(* CoDeSys 2.3.9.28 project: moje1.pro *)
(* Libraries: \\psf\Home\Documents\WAGO\libs\library\PowerMeasurement_01.lib 1.1.09 09:28:50, SysLibTime.lib 2.12.10 13:48:32, Building_common.lib 2.12.10 13:48:40, mod_com.lib 2.12.10 13:48:32, Util.lib 18.5.10 14:14:28, Standard.lib 2.12.10 13:48:34, SYSLIBCALLBACK.LIB 2.12.10 13:48:32, \\psf\Home\Documents\WAGO\libs\Libraries_BA\DALI_02.lib 4.3.11 14:50:14 *)

(* PLC configuration (modules and I/O channels)
TL01 AT %IX17.0 [BOOLOnX_I] Vypinac_sklad_sklad
TL02 AT %IX17.1 [BOOLOnX_I] Vypinac_sklad_prodejna
TL03 AT %IX17.2 [BOOLOnX_I] Vypinac_sklad_z_venku
TL04 AT %IX17.3 [BOOLOnX_I] Vypinac_sklad_vrata_predni
TL05 AT %IX17.4 [BOOLOnX_I] Vypinac_sklad_vrata_zadni
TL06 AT %IX17.5 [BOOLOnX_I] Vypinac_prodejna_kolotoc_sude
TL07 AT %IX17.6 [BOOLOnX_I] Vypinac_prodejna_kolotoc_liche
TL08 AT %IX17.7 [BOOLOnX_I] Vypinac_prodejna_vypinac
TL09 AT %IX17.8 [BOOLOnX_I] Prodejna_Dali
TL10 AT %IX17.9 [BOOLOnX_I] Prodejna_faugule_OUT13
TL11 AT %IX17.10 [BOOLOnX_I] Ch_3 Digital input
TL12 AT %IX17.11 [BOOLOnX_I] Ch_4 Digital input
TL13 AT %IX17.12 [BOOLOnX_I] Ch_5 Digital input
AT %IX17.13 [BOOLOnX_I] Ch_6 Digital input
AT %IX17.14 [BOOLOnX_I] Ch_7 Digital input
AT %IX17.15 [BOOLOnX_I] Ch_8 Digital input
0750-0430 8 DI 24 V DC 3.0ms [Type_1_8_Channels] node 2, in %IB2 out %QB2 {INTTypePAAssignment = PLC; INTTypeModule = plugged}
  AT %IX18.0 [BOOLOnX_I] Ch_1 Digital input
  AT %IX18.1 [BOOLOnX_I] Ch_2 Digital input
  AT %IX18.2 [BOOLOnX_I] Ch_3 Digital input
  AT %IX18.3 [BOOLOnX_I] Ch_4 Digital input
  AT %IX18.4 [BOOLOnX_I] Ch_5 Digital input
  AT %IX18.5 [BOOLOnX_I] Ch_6 Digital input
  AT %IX18.6 [BOOLOnX_I] Ch_7 Digital input
  AT %IX18.7 [BOOLOnX_I] Ch_8 Digital input
0750-0530 8 DO 24 V DC 0.5A [Type_10_8_Channels] node 3, in %IB3 out %QB3 {INTTypePAAssignment = PLC; INTTypeModule = plugged}
  KA01 AT %QX9.0 [BOOLOnX_Q] Nevim
  KA02 AT %QX9.1 [BOOLOnX_Q] kolotoc2
  KA03 AT %QX9.2 [BOOLOnX_Q] kolotoc3
  KA04 AT %QX9.3 [BOOLOnX_Q] kolotoc4
  KA05 AT %QX9.4 [BOOLOnX_Q] kolotoc5
  KA06 AT %QX9.5 [BOOLOnX_Q] kolotoc6
  KA07 AT %QX9.6 [BOOLOnX_Q] kolotoc7
  KA08 AT %QX9.7 [BOOLOnX_Q] kolotoc8
0750-0530 8 DO 24 V DC 0.5A [Type_10_8_Channels] node 4, in %IB4 out %QB4 {INTTypePAAssignment = PLC; INTTypeModule = plugged}
  KA09 AT %QX9.8 [BOOLOnX_Q] kolotoc9
  KA10 AT %QX9.9 [BOOLOnX_Q] kolotoc10
  KA11 AT %QX9.10 [BOOLOnX_Q] kolotoc11
  KA12 AT %QX9.11 [BOOLOnX_Q] kolotoc12
  KA13 AT %QX9.12 [BOOLOnX_Q] svetlo_vchod_do_prodejny
  KA14 AT %QX9.13 [BOOLOnX_Q] reklama
  KA15 AT %QX9.14 [BOOLOnX_Q] svetlo_vrata_predni
  KA16 AT %QX9.15 [BOOLOnX_Q] svetlo_vrata_zadni
0750-0530 8 DO 24 V DC 0.5A [Type_10_8_Channels] node 5, in %IB5 out %QB5 {INTTypePAAssignment = PLC; INTTypeModule = plugged}
  KA17 AT %QX10.0 [BOOLOnX_Q] Ch_1 Digital output
  AT %QX10.1 [BOOLOnX_Q] Ch_2 Digital output
  AT %QX10.2 [BOOLOnX_Q] Ch_3 Digital output
  KA20 AT %QX10.3 [BOOLOnX_Q] Ch_4 Digital output
  AT %QX10.4 [BOOLOnX_Q] Ch_5 Digital output
  AT %QX10.5 [BOOLOnX_Q] Ch_6 Digital output
  AT %QX10.6 [BOOLOnX_Q] Ch_7 Digital output
  AT %QX10.7 [BOOLOnX_Q] Ch_8 Digital output
0750-0530 8 DO 24 V DC 0.5A [Type_10_8_Channels] node 6, in %IB6 out %QB6 {INTTypePAAssignment = PLC; INTTypeModule = plugged}
  AT %QX10.8 [BOOLOnX_Q] Ch_1 Digital output
  AT %QX10.9 [BOOLOnX_Q] Ch_2 Digital output
  AT %QX10.10 [BOOLOnX_Q] Ch_3 Digital output
  AT %QX10.11 [BOOLOnX_Q] Ch_4 Digital output
  AT %QX10.12 [BOOLOnX_Q] Ch_5 Digital output
  AT %QX10.13 [BOOLOnX_Q] Ch_6 Digital output
  AT %QX10.14 [BOOLOnX_Q] Ch_7 Digital output
  AT %QX10.15 [BOOLOnX_Q] Ch_8 Digital output
Analog_1 AT %IW0 [WORDOnW_I] Ch_1 Input word
AT %IW1 [WORDOnW_I] Ch_2 Input word
AT %IW2 [WORDOnW_I] Ch_3 Input word
AT %IW3 [WORDOnW_I] Ch_4 Input word
Teplota_1 AT %IW4 [INTOnW_I] Ch_1 signed Input value
Teplota_2 AT %IW5 [INTOnW_I] Ch_2 signed Input value
Teplota_3 AT %IW6 [INTOnW_I] Ch_3 signed Input value
Teplota_4 AT %IW7 [INTOnW_I] Ch_4 signed Input value
0750-0641 DALI/DSI-Master [Type_36_1_Channels] node 9, in %IB9 out %QB9 {INTTypePAAssignment = PLC; INTTypeModule = plugged}
  AT %IX8.0 [BOOLOnX_I] Transmit accepted
  AT %IX8.1 [BOOLOnX_I] Receive request
  AT %IX8.2 [BOOLOnX_I] Init accepted
  AT %IX8.3 [BOOLOnX_I] Actor Error
  AT %IX8.4 [BOOLOnX_I] Frame Error
  AT %IX8.5 [BOOLOnX_I] Bus Error
  AT %IX8.6 [BOOLOnX_I] General Module Error
  AT %IB17 [BYTEOnB_I] DALI Response
  AT %IB18 [BYTEOnB_I] DALI Address
  AT %IB19 [BYTEOnB_I] Message 3
  AT %IB20 [BYTEOnB_I] Message 2
  AT %IB21 [BYTEOnB_I] Message 1
  AT %QX0.0 [BOOLOnX_Q] Transmit request
  AT %QX0.1 [BOOLOnX_Q] Receive accepted
  AT %QX0.2 [BOOLOnX_Q] Init request
  AT %QB1 [BYTEOnB_Q] DALI Command, DSI dimming value
  AT %QB2 [BYTEOnB_Q] DALI Address
  AT %QB3 [BYTEOnB_Q] Parameter 2
  AT %QB4 [BYTEOnB_Q] Parameter 1
  AT %QB5 [BYTEOnB_Q] Command extension
fazeVstup AT %IB22 [BYTEOnB_I] First Byte of 12
fazeVystup AT %QB6 [BYTEOnB_Q] First Byte of 12
Fieldbus variables [FB_VARS] node 1, in %IB0 out %QB0
*)

(* Task configuration *)
TASK hlavni (PRIORITY := 1, INTERVAL := T#20ms);
	PLC_PRG();
END_TASK

(* Global variable list: Global_Variables *)
VAR_GLOBAL
	start_bit: BOOL;
	Inicialiazace_DALI: BOOL;
	Inicializuj: BOOL;
	TL08s: BOOL;
	TL07s: BOOL;
	TL10s: BOOL;
	TL06s: BOOL;
	TL05s: BOOL;
	TL01s: BOOL;
	TL09s: BOOL;
	Cidlo: REAL;
	Uroven1: REAL := 3.5;
	Uroven2: REAL := 5;
	ZpozdeniCidla: BYTE := 10;
END_VAR

(* POU PLC_PRG, FBD *)
PROGRAM PLC_PRG
VAR
	cas_datum: CurTimeEx;
	System_cas: SysTime64;
	System_datum: SystemTimeDate;
	kolotoc1: kolotoc;
	kolotoc2: kolotoc;
	BLINK_nouzaky: BLINK;
	LibovolnyVystup: BOOL;
	kolo: KolotocF;
END_VAR
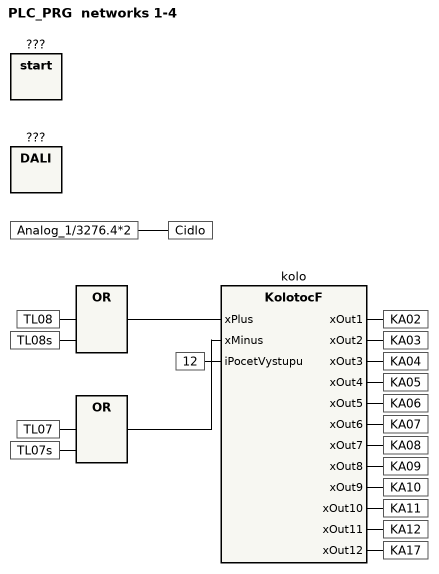
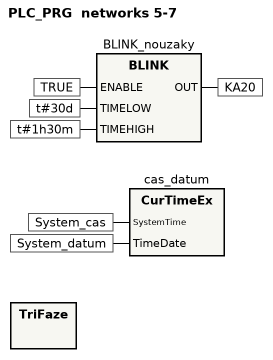
_FBD_ (* Function Block Diagram *)
NETWORK 1
	???:start()
NETWORK 2
	???:DALI()
NETWORK 3
	Analog_1/3276.4*2 => Cidlo
NETWORK 4
	kolo:KolotocF(xPlus: OR(TL08, TL08s), xMinus: OR(TL07, TL07s), iPocetVystupu: 12, xOut2 => KA03, xOut3 => KA04, xOut4 => KA05, xOut5 => KA06, xOut6 => KA07, xOut7 => KA08, xOut8 => KA09, xOut9 => KA10, xOut10 => KA11, xOut11 => KA12, xOut12 => KA17) => KA02
NETWORK 5
	BLINK_nouzaky:BLINK(ENABLE: TRUE, TIMELOW: t#30d, TIMEHIGH: t#1h30m) => KA20
NETWORK 6
	cas_datum:CurTimeEx(SystemTime: System_cas, TimeDate: System_datum)
NETWORK 7
	TriFaze()
_END_FBD_
(* the same logic as Structured Text *)
(* Network 1: see the listing above *)
(* Network 2: see the listing above *)
(* Network 3 *)
Cidlo := Analog_1/3276.4*2;
(* Network 4 *)
kolo(xPlus := TL08 OR TL08s, xMinus := TL07 OR TL07s, iPocetVystupu := 12);
KA03 := kolo.xOut2;
KA04 := kolo.xOut3;
KA05 := kolo.xOut4;
KA06 := kolo.xOut5;
KA07 := kolo.xOut6;
KA08 := kolo.xOut7;
KA09 := kolo.xOut8;
KA10 := kolo.xOut9;
KA11 := kolo.xOut10;
KA12 := kolo.xOut11;
KA17 := kolo.xOut12;
KA02 := kolo.xOut1;
(* Network 5 *)
BLINK_nouzaky(ENABLE := TRUE, TIMELOW := t#30d, TIMEHIGH := t#1h30m);
KA20 := BLINK_nouzaky.OUT;
(* Network 6 *)
cas_datum(SystemTime := System_cas, TimeDate := System_datum);
(* Network 7 *)
TriFaze();
END_PROGRAM

(* POU dali/kolotoc, FBD *)
FUNCTION_BLOCK kolotoc
VAR
	Data_platna: BOOL;
	Data_platna_reset: BOOL;
	T_Data_platna: TON;
	T_Data_platna_reset: TON;
	Stisk_kratky: BOOL := FALSE;
	Stisk_dlouhy: BOOL := FALSE;
	T_stisk_TLx: TON;
	F_trig_hr1: F_TRIG;
	R_trig_hr2: R_TRIG;
	TL1_Citac: CTU;
	SR_stisk_TLx: SR;
	ZAP_VYP: BOOL;




	TP_byl_kratky: TP;
	Q_byl_kratky: BOOL;
	blok_kratky: BOOL;
	TL1_hr1: BOOL;
	SET_stisk_TL1: BOOL;
	Q_stisk_TL1: BOOL;
	TL1_INT: INT;
END_VAR

VAR_OUTPUT
	Rele1: BOOL;
	Rele2: BOOL;
	Rele3: BOOL;
	Rele4: BOOL;
	Rele5: BOOL;
	Rele6: BOOL;
	Rele7: BOOL;
	Rele8: BOOL;
END_VAR
VAR_INPUT
	TL1: BOOL;
	RESET_Rezimu: BOOL;
	Pocet_rele: INT;
END_VAR
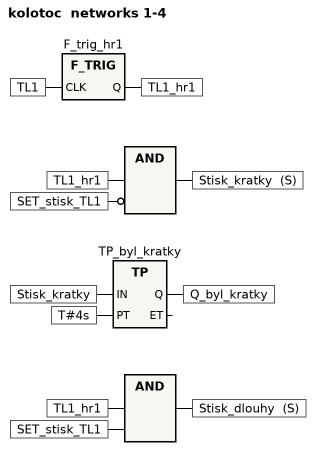
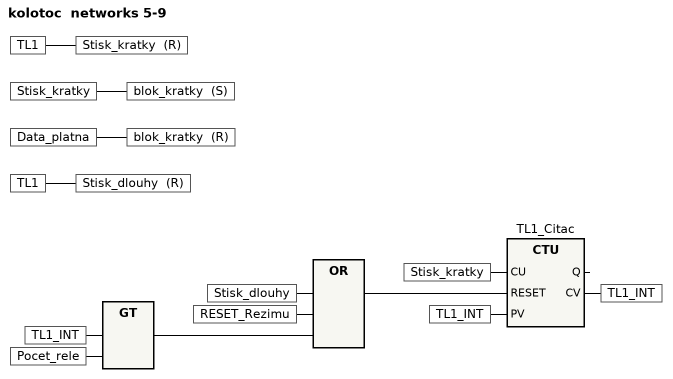
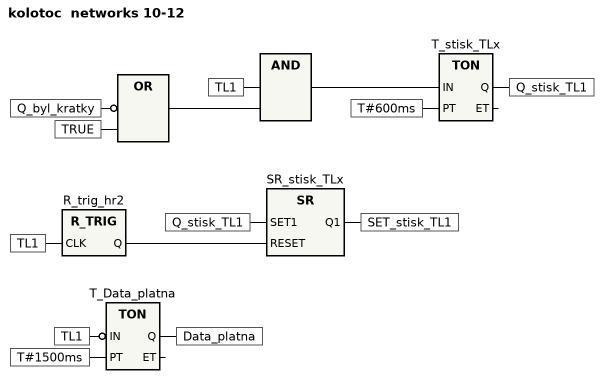
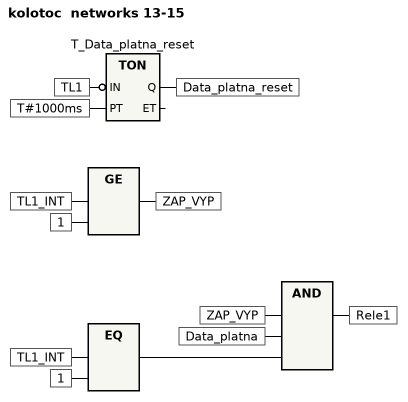
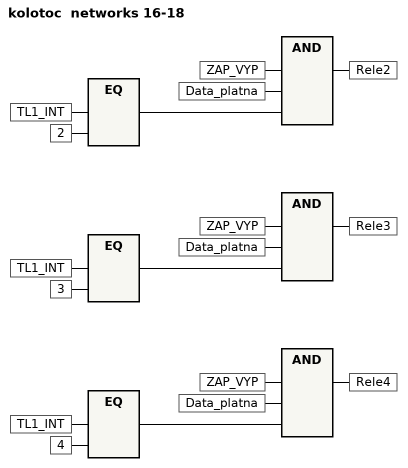
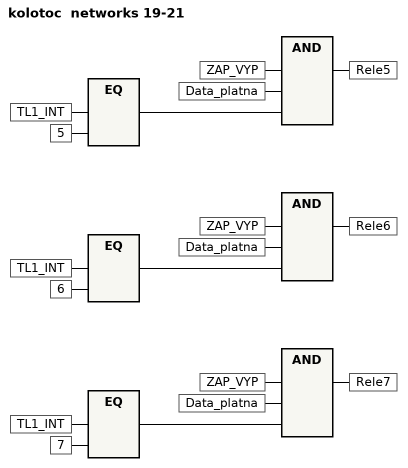
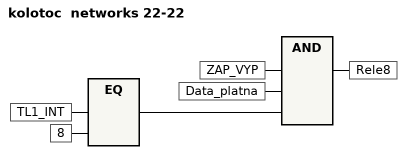
_FBD_ (* Function Block Diagram *)
NETWORK 1
	F_trig_hr1:F_TRIG(CLK: TL1) => TL1_hr1
NETWORK 2
	AND(TL1_hr1, NOT SET_stisk_TL1) => S Stisk_kratky
NETWORK 3
	TP_byl_kratky:TP(IN: Stisk_kratky, PT: T#4s) => Q_byl_kratky
NETWORK 4
	AND(TL1_hr1, SET_stisk_TL1) => S Stisk_dlouhy
NETWORK 5
	TL1 => R Stisk_kratky
NETWORK 6
	Stisk_kratky => S blok_kratky
NETWORK 7
	Data_platna => R blok_kratky
NETWORK 8
	TL1 => R Stisk_dlouhy
NETWORK 9
	TL1_Citac:CTU(CU: Stisk_kratky, RESET: OR(Stisk_dlouhy, RESET_Rezimu, GT(TL1_INT, Pocet_rele)), PV: TL1_INT, CV => TL1_INT)
NETWORK 10 (* delka stisku TLx *)
	T_stisk_TLx:TON(IN: AND(TL1, OR(NOT Q_byl_kratky, TRUE)), PT: T#600ms) => Q_stisk_TL1
NETWORK 11
	SR_stisk_TLx:SR(SET1: Q_stisk_TL1, RESET: R_trig_hr2:R_TRIG(CLK: TL1)) => SET_stisk_TL1
NETWORK 12 (* Data platna *)
	T_Data_platna:TON(IN: NOT TL1, PT: T#1500ms) => Data_platna
NETWORK 13 (* Data platna *)
	T_Data_platna_reset:TON(IN: NOT TL1, PT: T#1000ms) => Data_platna_reset
NETWORK 14
	GE(TL1_INT, 1) => ZAP_VYP
NETWORK 15
	AND(ZAP_VYP, Data_platna, EQ(TL1_INT, 1)) => Rele1
NETWORK 16
	AND(ZAP_VYP, Data_platna, EQ(TL1_INT, 2)) => Rele2
NETWORK 17
	AND(ZAP_VYP, Data_platna, EQ(TL1_INT, 3)) => Rele3
NETWORK 18
	AND(ZAP_VYP, Data_platna, EQ(TL1_INT, 4)) => Rele4
NETWORK 19
	AND(ZAP_VYP, Data_platna, EQ(TL1_INT, 5)) => Rele5
NETWORK 20
	AND(ZAP_VYP, Data_platna, EQ(TL1_INT, 6)) => Rele6
NETWORK 21
	AND(ZAP_VYP, Data_platna, EQ(TL1_INT, 7)) => Rele7
NETWORK 22
	AND(ZAP_VYP, Data_platna, EQ(TL1_INT, 8)) => Rele8
_END_FBD_
(* the same logic as Structured Text *)
(* Network 1 *)
F_trig_hr1(CLK := TL1);
TL1_hr1 := F_trig_hr1.Q;
(* Network 2 *)
IF TL1_hr1 AND NOT SET_stisk_TL1 THEN Stisk_kratky := TRUE; END_IF;
(* Network 3 *)
TP_byl_kratky(IN := Stisk_kratky, PT := T#4s);
Q_byl_kratky := TP_byl_kratky.Q;
(* Network 4 *)
IF TL1_hr1 AND SET_stisk_TL1 THEN Stisk_dlouhy := TRUE; END_IF;
(* Network 5 *)
IF TL1 THEN Stisk_kratky := FALSE; END_IF;
(* Network 6 *)
IF Stisk_kratky THEN blok_kratky := TRUE; END_IF;
(* Network 7 *)
IF Data_platna THEN blok_kratky := FALSE; END_IF;
(* Network 8 *)
IF TL1 THEN Stisk_dlouhy := FALSE; END_IF;
(* Network 9 *)
TL1_Citac(CU := Stisk_kratky, RESET := Stisk_dlouhy OR RESET_Rezimu OR (TL1_INT > Pocet_rele), PV := TL1_INT);
TL1_INT := TL1_Citac.CV;
(* Network 10: see the listing above *)
(* Network 11 *)
R_trig_hr2(CLK := TL1);
SR_stisk_TLx(SET1 := Q_stisk_TL1, RESET := R_trig_hr2.Q);
SET_stisk_TL1 := SR_stisk_TLx.Q1;
(* Network 12 *)
T_Data_platna(IN := NOT TL1, PT := T#1500ms);
Data_platna := T_Data_platna.Q;
(* Network 13 *)
T_Data_platna_reset(IN := NOT TL1, PT := T#1000ms);
Data_platna_reset := T_Data_platna_reset.Q;
(* Network 14 *)
ZAP_VYP := TL1_INT >= 1;
(* Network 15 *)
Rele1 := ZAP_VYP AND Data_platna AND (TL1_INT = 1);
(* Network 16 *)
Rele2 := ZAP_VYP AND Data_platna AND (TL1_INT = 2);
(* Network 17 *)
Rele3 := ZAP_VYP AND Data_platna AND (TL1_INT = 3);
(* Network 18 *)
Rele4 := ZAP_VYP AND Data_platna AND (TL1_INT = 4);
(* Network 19 *)
Rele5 := ZAP_VYP AND Data_platna AND (TL1_INT = 5);
(* Network 20 *)
Rele6 := ZAP_VYP AND Data_platna AND (TL1_INT = 6);
(* Network 21 *)
Rele7 := ZAP_VYP AND Data_platna AND (TL1_INT = 7);
(* Network 22 *)
Rele8 := ZAP_VYP AND Data_platna AND (TL1_INT = 8);
END_FUNCTION_BLOCK

(* POU Kolotoc/KolotocF, CFC *)
FUNCTION_BLOCK KolotocF
VAR
END_VAR
VAR_INPUT
	xPlus: BOOL;
	xMinus: BOOL;
	iPocetVystupu: INT;
END_VAR
VAR_OUTPUT
	xOut1: BOOL;
	xOut2: BOOL;
	xOut3: BOOL;
	xOut4: BOOL;
	xOut5: BOOL;
	xOut6: BOOL;
	xOut7: BOOL;
	xOut8: BOOL;
	xOut9: BOOL;
	xOut10: BOOL;
	xOut11: BOOL;
	xOut12: BOOL;
END_VAR
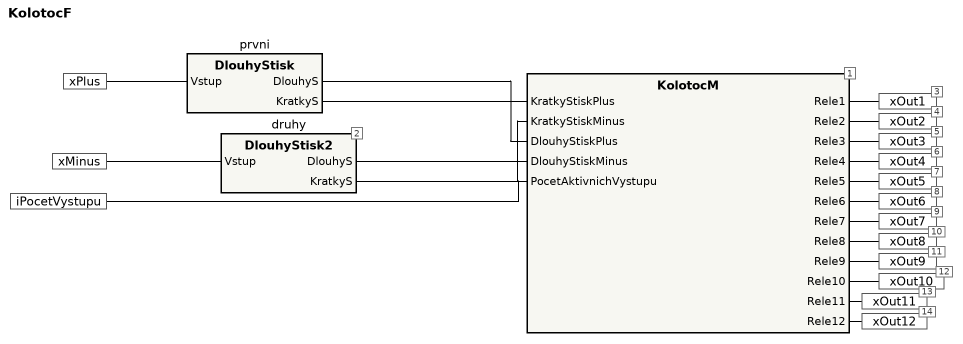
_CFC_ (* Continuous Function Chart, elements in execution order *)
#0 prvni:DlouhyStisk(Vstup: xPlus)
#1 KolotocM(KratkyStiskPlus: #0.KratkyS, KratkyStiskMinus: #2.KratkyS, DlouhyStiskPlus: #0.DlouhyS, DlouhyStiskMinus: #2.DlouhyS, PocetAktivnichVystupu: iPocetVystupu)
#2 druhy:DlouhyStisk2(Vstup: xMinus)
#3 xOut1 <= #1.Rele1
#4 xOut2 <= #1.Rele2
#5 xOut3 <= #1.Rele3
#6 xOut4 <= #1.Rele4
#7 xOut5 <= #1.Rele5
#8 xOut6 <= #1.Rele6
#9 xOut7 <= #1.Rele7
#10 xOut8 <= #1.Rele8
#11 xOut9 <= #1.Rele9
#12 xOut10 <= #1.Rele10
#13 xOut11 <= #1.Rele11
#14 xOut12 <= #1.Rele12
_END_CFC_
(* the same logic as Structured Text *)
prvni(Vstup := xPlus);
KolotocM(KratkyStiskPlus := prvni.KratkyS, KratkyStiskMinus := druhy.KratkyS, DlouhyStiskPlus := prvni.DlouhyS, DlouhyStiskMinus := druhy.DlouhyS, PocetAktivnichVystupu := iPocetVystupu);
druhy(Vstup := xMinus);
xOut1 := KolotocM.Rele1;
xOut2 := KolotocM.Rele2;
xOut3 := KolotocM.Rele3;
xOut4 := KolotocM.Rele4;
xOut5 := KolotocM.Rele5;
xOut6 := KolotocM.Rele6;
xOut7 := KolotocM.Rele7;
xOut8 := KolotocM.Rele8;
xOut9 := KolotocM.Rele9;
xOut10 := KolotocM.Rele10;
xOut11 := KolotocM.Rele11;
xOut12 := KolotocM.Rele12;
END_FUNCTION_BLOCK

(* POU Kolotoc/DlouhyStisk, CFC *)
PROGRAM DlouhyStisk
VAR_INPUT
	Vstup: BOOL;
END_VAR
VAR_OUTPUT
	DlouhyS: BOOL;
	KratkyS: BOOL;
END_VAR
VAR
	cas1: TON;
	cas2: TOF;
	cas3: TON;
	cas4: TOF;
END_VAR
VAR (* helpers for the ST form of the networks *)
	_t57 : BOOL;
END_VAR
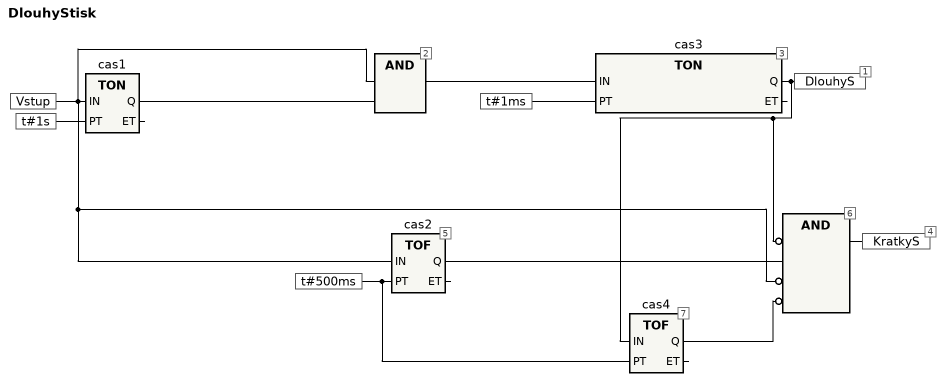
_CFC_ (* Continuous Function Chart, elements in execution order *)
#0 cas1:TON(IN: Vstup, PT: t#1s)
#1 DlouhyS <= #3.Q
#2 AND(Vstup, #0.Q)
#3 cas3:TON(IN: #2, PT: t#1ms)
#4 KratkyS <= #6
#5 cas2:TOF(IN: Vstup, PT: t#500ms)
#6 AND(NOT #3.Q, #5.Q, NOT Vstup, NOT #7.Q)
#7 cas4:TOF(IN: #3.Q, PT: t#500ms)
_END_CFC_
(* the same logic as Structured Text *)
cas1(IN := Vstup, PT := t#1s);
DlouhyS := cas3.Q;
cas3(IN := Vstup AND cas1.Q, PT := t#1ms);
KratkyS := _t57;
cas2(IN := Vstup, PT := t#500ms);
_t57 := NOT cas3.Q AND cas2.Q AND NOT Vstup AND NOT cas4.Q;
cas4(IN := cas3.Q, PT := t#500ms);
END_PROGRAM

(* POU Kolotoc/KolotocM, ST *)
PROGRAM KolotocM
VAR
	index: INT := 0;
	a: BOOL := FALSE;
	b: BOOL := FALSE;
END_VAR
VAR_INPUT
	KratkyStiskPlus: BOOL;
	KratkyStiskMinus: BOOL;
	DlouhyStiskPlus: BOOL;
	DlouhyStiskMinus: BOOL;
	PocetAktivnichVystupu: INT;
END_VAR
VAR_OUTPUT
	Rele1: BOOL;
	Rele2: BOOL;
	Rele3: BOOL;
	Rele4: BOOL;
	Rele5: BOOL;
	Rele6: BOOL;
	Rele7: BOOL;
	Rele8: BOOL;
	Rele9: BOOL;
	Rele10: BOOL;
	Rele11: BOOL;
	Rele12: BOOL;
END_VAR
IF (KratkyStiskPlus)
THEN
	a := TRUE;
END_IF

IF (a AND KratkyStiskPlus = FALSE)
	THEN
	index := index + 1;
	a := FALSE;
END_IF

IF (KratkyStiskMinus)
THEN
	b := TRUE;
END_IF

IF (b AND KratkyStiskMinus = FALSE)
THEN
	index := index - 1;
	b := FALSE;
END_IF

IF (index = -1)
THEN
	index := PocetAktivnichVystupu;
END_IF

IF (index = PocetAktivnichVystupu + 1)
THEN
	index := 0;
END_IF

IF (index = 0 )
THEN
	Rele1 := FALSE;
	Rele2 := FALSE;
	Rele3 := FALSE;
	Rele4 := FALSE;
	Rele5 := FALSE;
	Rele6 := FALSE;
	Rele7 := FALSE;
	Rele8 := FALSE;
	Rele9 := FALSE;
	Rele10 := FALSE;
	Rele11 := FALSE;
	Rele12 := FALSE;
ELSIF (index = 1)
THEN
	Rele1 := TRUE;
	Rele2 := FALSE;
	Rele3 := FALSE;
	Rele4 := FALSE;
	Rele5 := FALSE;
	Rele6 := FALSE;
	Rele7 := FALSE;
	Rele8 := FALSE;
	Rele9 := FALSE;
	Rele10 := FALSE;
ELSIF (index = 2)
THEN
	Rele1 := FALSE;
	Rele2 := TRUE;
	Rele3 := FALSE;
	Rele4 := FALSE;
	Rele5 := FALSE;
	Rele6 := FALSE;
	Rele7 := FALSE;
	Rele8 := FALSE;
	Rele9 := FALSE;
	Rele10 := FALSE;
	Rele11 := FALSE;
	Rele12 := FALSE;
ELSIF (index = 3)
THEN
	Rele1 := FALSE;
	Rele2 := FALSE;
	Rele3 := TRUE;
	Rele4 := FALSE;
	Rele5 := FALSE;
	Rele6 := FALSE;
	Rele7 := FALSE;
	Rele8 := FALSE;
	Rele9 := FALSE;
	Rele10 := FALSE;
	Rele11 := FALSE;
	Rele12 := FALSE;
ELSIF (index = 4)
THEN
	Rele1 := FALSE;
	Rele2 := FALSE;
	Rele3 := FALSE;
	Rele4 := TRUE;
	Rele5 := FALSE;
	Rele6 := FALSE;
	Rele7 := FALSE;
	Rele8 := FALSE;
	Rele9 := FALSE;
	Rele10 := FALSE;
	Rele11 := FALSE;
	Rele12 := FALSE;
ELSIF (index = 5)
THEN
	Rele1 := FALSE;
	Rele2 := FALSE;
	Rele3 := FALSE;
	Rele4 := FALSE;
	Rele5 := TRUE;
	Rele6 := FALSE;
	Rele7 := FALSE;
	Rele8 := FALSE;
	Rele9 := FALSE;
	Rele10 := FALSE;
	Rele11 := FALSE;
	Rele12 := FALSE;
ELSIF (index = 6)
THEN
	Rele1 := FALSE;
	Rele2 := FALSE;
	Rele3 := FALSE;
	Rele4 := FALSE;
	Rele5 := FALSE;
	Rele6 := TRUE;
	Rele7 := FALSE;
	Rele8 := FALSE;
	Rele9 := FALSE;
	Rele10 := FALSE;
	Rele11 := FALSE;
	Rele12 := FALSE;
ELSIF (index = 7)
THEN
	Rele1 := FALSE;
	Rele2 := FALSE;
	Rele3 := FALSE;
	Rele4 := FALSE;
	Rele5 := FALSE;
	Rele6 := FALSE;
	Rele7 := TRUE;
	Rele8 := FALSE;
	Rele9 := FALSE;
	Rele10 := FALSE;
	Rele11 := FALSE;
	Rele12 := FALSE;
ELSIF (index = 8)
THEN
	Rele1 := FALSE;
	Rele2 := FALSE;
	Rele3 := FALSE;
	Rele4 := FALSE;
	Rele5 := FALSE;
	Rele6 := FALSE;
	Rele7 := FALSE;
	Rele8 := TRUE;
	Rele9 := FALSE;
	Rele10 := FALSE;
	Rele11 := FALSE;
	Rele12 := FALSE;
ELSIF (index = 9)
THEN
	Rele1 := FALSE;
	Rele2 := FALSE;
	Rele3 := FALSE;
	Rele4 := FALSE;
	Rele5 := FALSE;
	Rele6 := FALSE;
	Rele7 := FALSE;
	Rele8 := FALSE;
	Rele9 := TRUE;
	Rele10 := FALSE;
	Rele11 := FALSE;
	Rele12 := FALSE;
ELSIF (index = 10)
THEN
	Rele1 := FALSE;
	Rele2 := FALSE;
	Rele3 := FALSE;
	Rele4 := FALSE;
	Rele5 := FALSE;
	Rele6 := FALSE;
	Rele7 := FALSE;
	Rele8 := FALSE;
	Rele9 := FALSE;
	Rele10 := TRUE;
	Rele11 := FALSE;
	Rele12 := FALSE;
ELSIF (index = 11)
THEN
	Rele1 := FALSE;
	Rele2 := FALSE;
	Rele3 := FALSE;
	Rele4 := FALSE;
	Rele5 := FALSE;
	Rele6 := FALSE;
	Rele7 := FALSE;
	Rele8 := FALSE;
	Rele9 := FALSE;
	Rele10 := FALSE;
	Rele11 := TRUE;
	Rele12 := FALSE;
ELSIF (index = 12)
THEN
	Rele1 := FALSE;
	Rele2 := FALSE;
	Rele3 := FALSE;
	Rele4 := FALSE;
	Rele5 := FALSE;
	Rele6 := FALSE;
	Rele7 := FALSE;
	Rele8 := FALSE;
	Rele9 := FALSE;
	Rele10 := FALSE;
	Rele11 := FALSE;
	Rele12 := TRUE;
END_IF
IF (DlouhyStiskPlus)
THEN
	index := 0;
END_IF

IF (DlouhyStiskMinus)
THEN
	index := 0;
END_IF
END_PROGRAM

(* POU Kolotoc/DlouhyStisk2, CFC *)
PROGRAM DlouhyStisk2
VAR_INPUT
	Vstup: BOOL;
END_VAR
VAR_OUTPUT
	DlouhyS: BOOL;
	KratkyS: BOOL;
END_VAR
VAR
	cas1: TON;
	cas2: TOF;
	cas3: TON;
	cas4: TOF;
END_VAR
VAR (* helpers for the ST form of the networks *)
	_t57 : BOOL;
END_VAR
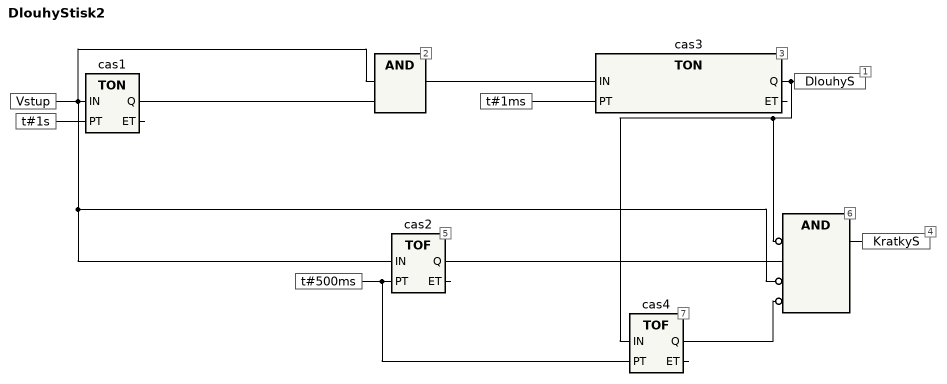
_CFC_ (* Continuous Function Chart, elements in execution order *)
#0 cas1:TON(IN: Vstup, PT: t#1s)
#1 DlouhyS <= #3.Q
#2 AND(Vstup, #0.Q)
#3 cas3:TON(IN: #2, PT: t#1ms)
#4 KratkyS <= #6
#5 cas2:TOF(IN: Vstup, PT: t#500ms)
#6 AND(NOT #3.Q, #5.Q, NOT Vstup, NOT #7.Q)
#7 cas4:TOF(IN: #3.Q, PT: t#500ms)
_END_CFC_
(* the same logic as Structured Text *)
cas1(IN := Vstup, PT := t#1s);
DlouhyS := cas3.Q;
cas3(IN := Vstup AND cas1.Q, PT := t#1ms);
KratkyS := _t57;
cas2(IN := Vstup, PT := t#500ms);
_t57 := NOT cas3.Q AND cas2.Q AND NOT Vstup AND NOT cas4.Q;
cas4(IN := cas3.Q, PT := t#500ms);
END_PROGRAM

(* POU start, FBD *)
PROGRAM start
VAR
END_VAR
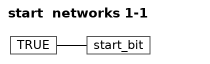
_FBD_ (* Function Block Diagram *)
NETWORK 1
	TRUE => start_bit
_END_FBD_
(* the same logic as Structured Text *)
(* Network 1 *)
start_bit := TRUE;
END_PROGRAM

(* POU dali/DALI, FBD *)
PROGRAM DALI
VAR
	trojklik_sklad: Trojklik;
	D_M: FbDALI_Joblist;

	Jobs: typDaliJoblisten;
	short_group: BOOL := FALSE;
	hodnota_po_zapnuti: BYTE := 50;
	hodnota_po_zapnuti_prodejna: BYTE := 100;
	povolit_vypnuti_pri_minimum: BOOL := FALSE;
	rychlost_zneny: BYTE := 7;
	co_je_kratky_a_dlouhy_stisk: TIME := t#600ms;
      OP_reset1: BOOL;
	OP_reset2: BOOL;
	OP_reset3: BOOL;
	OP_reset_OUT15: BOOL;
	OP_reset_OUT16: BOOL;

	Svetlo_adr1: FbDALI_LatchingRelay;
	Svetlo_adr2: FbDALI_LatchingRelay;
	Svetlo_adr3: FbDALI_LatchingRelay;
	Svetlo_adr4: FbDALI_DimmSingleButton;

	stav_adr1: BYTE;
	stav_adr2: BYTE;
	stav_adr3: BYTE;
	stav_adr4: BYTE;


	trojklik_prodejna: Trojklik;
	OP_reset4: BOOL;
	Trojklik_Fagule_OUT13: Trojklik;
	OP_reset5: BOOL;
	TP_ALL: TP;
	Q_All: BOOL;
	Dali_Status_03: FbDALI_StatusDimmValue;
	dali_status_Ready03: BOOL;
	dali_status_Feedback03: BYTE;
	dali_status_Status03: BOOL;
	dali_DimmValue_Ready03: BYTE;
	Reset_ini: TON;
	Dali_Status_09: FbDALI_StatusDimmValue;
	dali_status_Ready09: BOOL;
	dali_status_Feedback09: BYTE;
	dali_status_Status09: BOOL;
	dali_DimmValue_Ready09: BYTE;
	Dali_Status_19: FbDALI_StatusDimmValue;
	dali_status_Ready19: BOOL;
	dali_status_Feedback19: BYTE;
	dali_status_Status19: BOOL;
	dali_DimmValue_Ready19: BYTE;
	TON_ALL: TON;
	pom1: BOOL;
	go: BOOL;


	Fb_ShortLong1: Fb_ShortLong;
	CTU1: CTU;
	R_TRIG1: R_TRIG;
	TP1: TP;
	F_TRIG1: F_TRIG;
	STAV: WORD;
	CasNaKlik: TIME := t#1s500ms;
	F_TRIG2: F_TRIG;
	R_TRIG2: R_TRIG;
	Zhasni1: Zhasni;
	F_TRIG3: F_TRIG;
	Fb_LatchingRelay1: Fb_LatchingRelay;
	KratkyKlik: BOOL;
	Fb_ShortLong2: Fb_ShortLong;
	Fb_LatchingRelay2: Fb_LatchingRelay;
	Fb_ShortLong3: Fb_ShortLong;
	KratkyKlikA: BOOL;
	KratkyKlikB: BOOL;
	KratkyKlikC: BOOL;
	Svetlo_adr_255: FbDALI_LatchingRelay;
	stav_adr255: BYTE;
	TON_Cental_Off: TON;
	R_TRIG6: R_TRIG;
	ka15cas: TON;
	ka15pink: TP;
	TL06p: BOOL;
	ka16cas: TON;
	ka16pink: TP;
	TL05p: BOOL;
	ka13cas: TON;
	ka13pink: TP;
 	TL10p: BOOL;
	casvensvetel: TIME:= t#10m;
	Svetlo_adr5: FbDALI_LatchingRelay;
	stav_adr5: BYTE;
	Svetlo_adr6: FbDALI_LatchingRelay;
	stav_adr6: BYTE;
	Ovladani: Ovladani_7_8_9;
	aaa: BOOL;
	Svetlo_adr7: FbDALI_LatchingRelay;
	stav_adr7: BYTE;
	Svetlo_adr8: FbDALI_LatchingRelay;
	stav_adr8: BYTE;
	Svetlo_adr9: FbDALI_LatchingRelay;
	stav_adr9: BYTE;
END_VAR
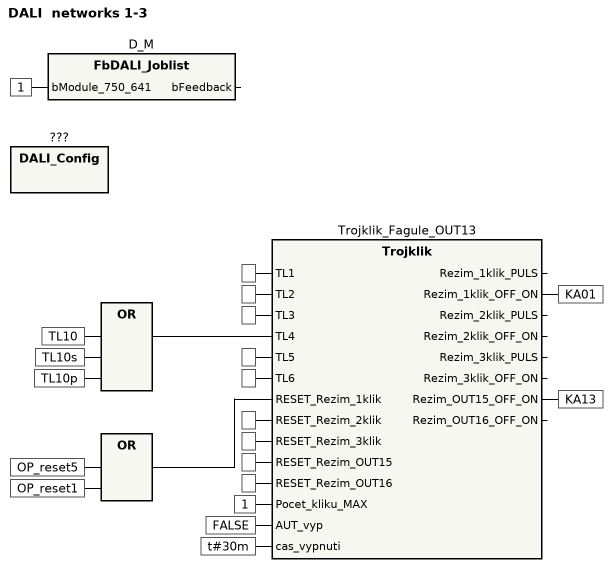
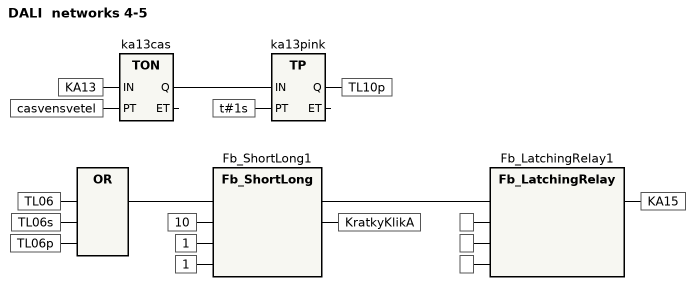
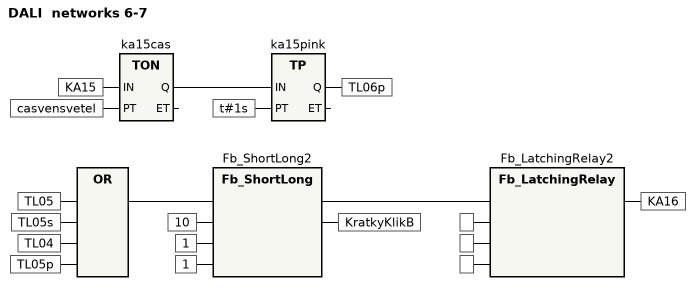
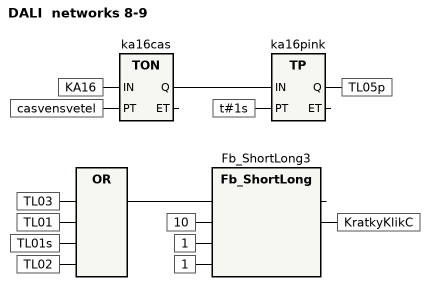
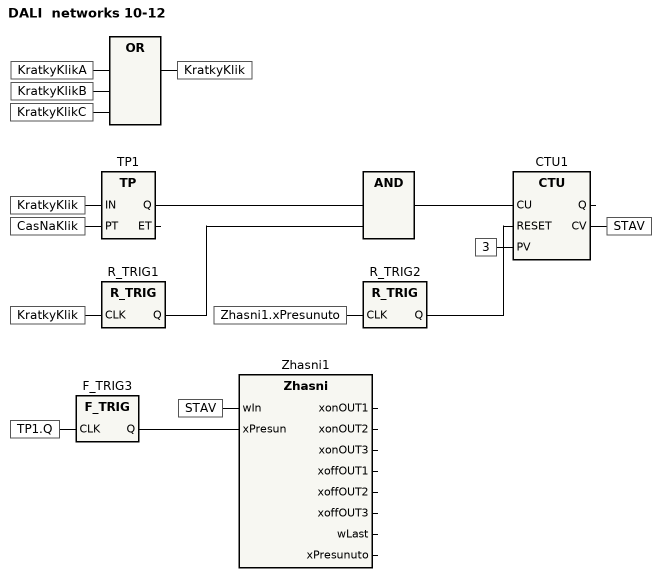
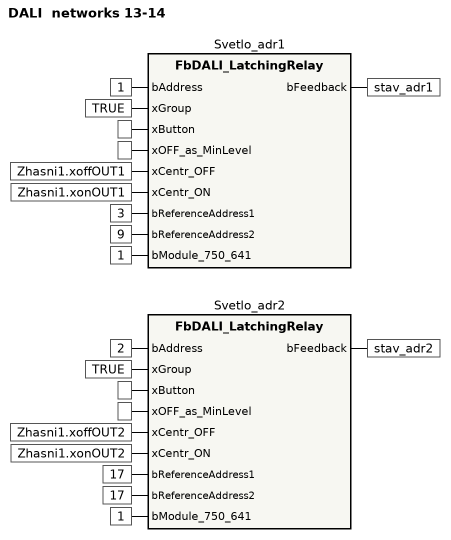
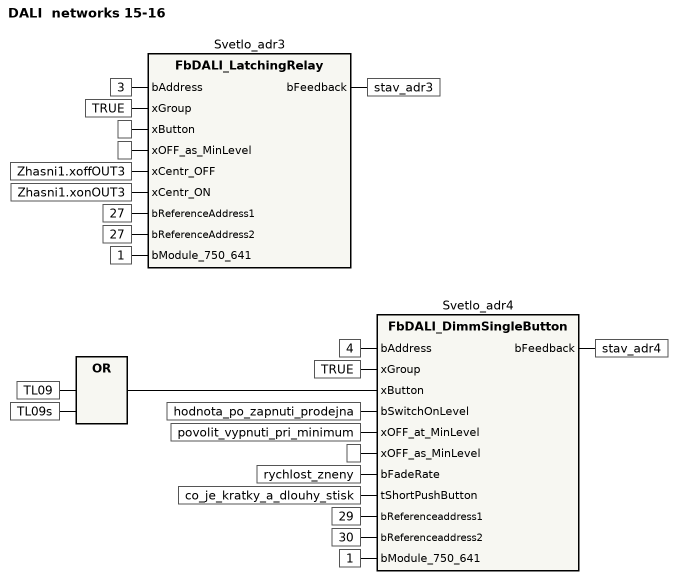
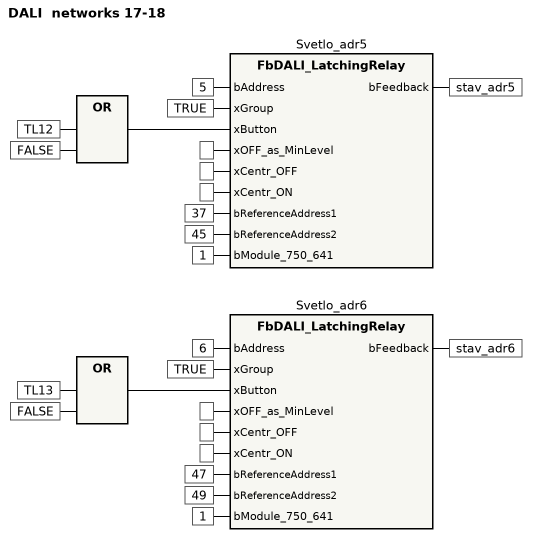
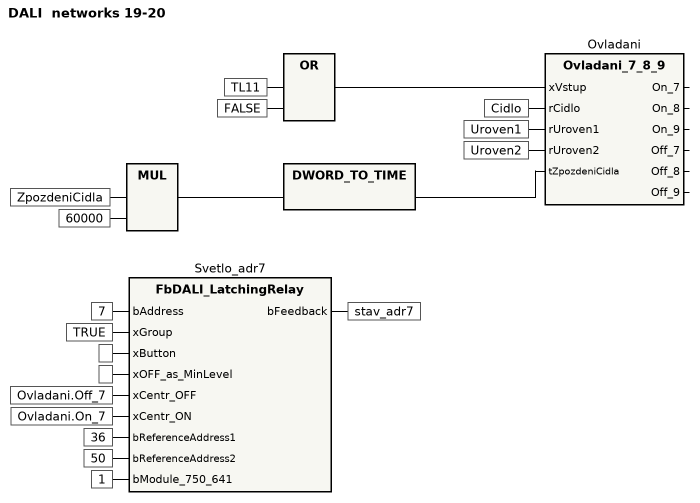
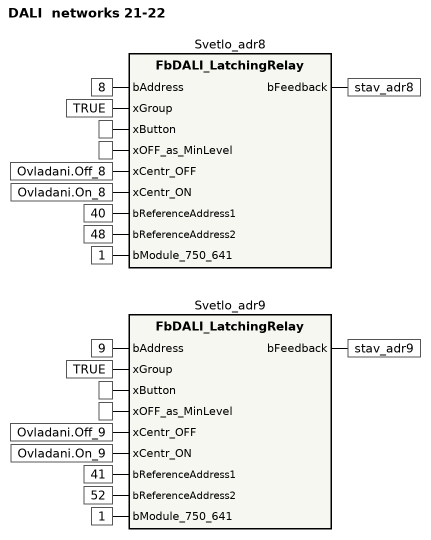
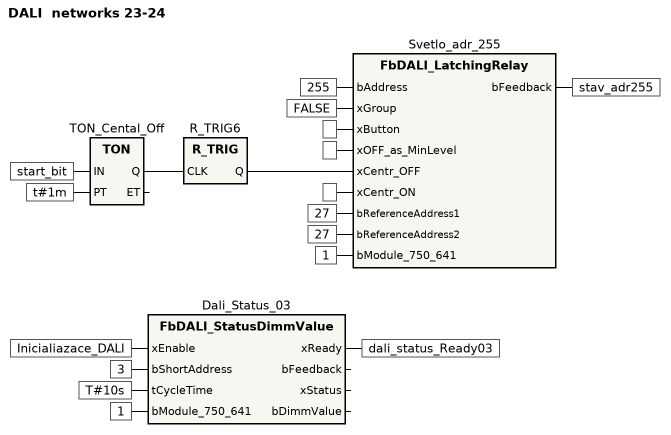
